# EPICS autosave request: CARS/iocBoot/iocDCM/auto_settings.req
file XFM_motor_settings.req",  P=$(P), M=m1
file XFM_motor_settings.req",  P=$(P), M=m2
file XFM_motor_settings.req",  P=$(P), M=m3
file XFM_motor_settings.req",  P=$(P), M=m4
file XFM_motor_settings.req",  P=$(P), M=m5
